FUNCTION F_SetExternalGroupError : BOOL
(**************************************************************************************
 * 	Application		:	BoxControl Framework
 *	Revision		:	$Revision: 404529 $
 *	Revision date	:	$Date: 2018-04-23 08:21:38 +0200 (Mo., 23 Apr 2018) $
 *	Last changed by	:	$Author: b7bolm $
 *	URL				:	$URL: http://almscdc.swisslog.com/repo/SWPD/Development/BoxControlFramework/20_Release/trunk/01_Software/BCF/BCF/JumpStart/20_Product/10_App/14_Groups/10_Lib/10_Conv/10_Functions/F_SetExternalGroupError.TcPOU $
 *
 *	Purpose			:	Set external error
 *						Add an External error, which will be reported over the configured
 *						position.
 *						
 *
 * ------------------------------------------------------------------------------------
 *	Copyright Swisslog [IP AG], Switzerland. All rights reserved.
 * 
 * ------------------------------------------------------------------------------------
 *	
 * 	Revision History: 
 *
 * 	VERSION			DATE			INITIALS			DESCRIPTION
 *	0.1				01.01.2001		swl					Example
 *
 **************************************************************************************)
VAR_INPUT
	eGroupNumber	: E_GroupNumber;
	ErrorType		: E_ErrorType; // Error message type
	ErrorParam		: STRING(System.ERROR_PARAM_STRINGLENGTH); // Error parameter
	ErrorMsg		: INT; // Error message as String (Will be mapped to error code)
END_VAR


// Validate inputs
IF eGroupNumber >  E_GroupNumber.G_BEGIN_GROUP THEN
	IF __ISVALIDREF(GroupRegistry[eGroupNumber].rGroup) THEN
		// Set external error on instance
		GroupRegistry[eGroupNumber].rGroup.M_SetExternalError(
			mErrorType 	:= ErrorType,
			mErrorParam := ErrorParam,
			mErrorCode 	:= ErrorMsg);
	END_IF
END_IF

END_FUNCTION

(* stored: Version 1.1.0.1, ProductVersion 3.1.4022.12
   POU F_SetExternalGroupError: Id {096762a6-6a65-4897-a2db-2de473f16d30}, SpecialFunc None *)
